# B&R Automation Studio project CleanChemi_SiteManagementSystem
Automation Studio 4.12.7.113 SP; technology packages: mapp 5.24.3, mappView 5.24.4

## Configuration 1584

### Task classes (Cpu.sw)
```
Cyclic#1 (cycle 50000 us, tolerance 50000 us):
  ModMaster <- modbusTCP.ModMaster.prg
  Main <- Main.prg
  ModbusDriv <- (binary)
Cyclic#2 (cycle 100000 us, tolerance 100000 us):
  Vis <- Vis.prg
Cyclic#4:
  Services <- Services.prg
DataObjects: Acp10sys
Binaries: FWRules, TCData, mvLoader, udbdef, TCLang, acp10cfg, arnc0cfg, Acp10map, iomap, arconfig, asfw, ashwac, sysconf, User, Role, ashwd, TC
Libraries: AsOpcUas, AsOpcUac, runtime, NcGlobal, standard, MbusTCP, IDEC_Real, astime, AsIecCon, AsTCP, AsBrStr, AsARCfg, sys_lib, ArTextSys, Str2DtPvdr, powerlnk, arssl, asstring, AsBrWStr, MpCom, MpBase, HA, HA_Version, HA_IO, HA_Dir, HA_Convert, HA_Str, HA_AlarmX, HA_ItemX, HA_RAND, ArEventLog, ArProject, brsystem, FileIO, AsUSB, HA_Array, HA_SysErr, MpAlarmX, IDEC_Strng, MpUserX, AsHttp, AsICMP, AsHost
```

### Hardware
```
X20CP1584 : X20CP1584 v1.10.0.0
  Connector IF1:
    ActivateIna = 0
  Connector IF2:
    ActivateDevice = 1
    Mode = Manual
    InternetAddress = 172.16.1.63
    SubnetMask = 255.255.255.0
    InaPort = 11160
    ActivateSnmp = 2
    ActivateModbus = 1
    NumSlaves = -1
    NumAllBlocks = -1
    MemSizeIn = -1
    MemSizeOut = -1
    SlaveDiagnostics = 1
  ConfigurationID = RemoteVis_CleanChemistry_Config1
  VolatileGlobalPvSize = 6553500
  SystemTick = 10000
  TaskClassIdleTime = 10000
  Cyclic1Duration = 50000
  Cyclic1Tolerance = 50000
  Cyclic2Duration = 100000
  Cyclic2Tolerance = 100000
  FileDevice1
  FileDeviceName1 = USER_DEVICE
  FileDevicePath1 = F:\
  FileDevice2
  FileDeviceName2 = USER_DEVICE_SIM
  FileDevicePath2 = ..\..\..\..\USER_DEVICE\
  EthernetDefaultGateway = 172.16.1.62
  ActivateDns = 1
  DnsServer1 = 8.8.8.8
  FtpUser1
  FtpUsername1 = brcpu
  FtpUserPassword1 = 20s6X0g3G25vRkBYChW+IYrxlgFH8I/njpAQzwadF+E=  // brcpu
  FtpUserSalt1 = aGb711uD
  FTPAccessRight1 = 0
  FTPdevice1 = ALL
  ActivateOpcUa = 1
  OpcUaInformationModels_PV_Version = 1
```

### Config_2.mpalarmxhistory - X20CP1584/mappServices/Config_2.mpalarmxhistory
```
Element gAlarmXHistory (Type=mpalarmxhistory)
  mapp.AlarmX.History:
    Export:
      FileNamePattern = AlarmHistory/Alarms_%Y_%m_%d_%H_%M_%S.csv
    Memory:
      MemorySize = 5
      BufferSize = 1
      MemoryType = 3
```

### Config_3.mpuserx - X20CP1584/mappServices/Config_3.mpuserx
```
Element UserMgmtX (Type=mpuserx)
  UserMgmtSystem:
    UserMgmtSystemType = 1
  ServerSettings:
    Server:
      AdditionalUserData:
        [0] = mail
        [1] = telephoneNumber
```

## Configuration 3100

CPU 5APC3100.KBU3-000, AutomationRuntime Q4.93, Build 4.1.2, Safety 0.0, Vc 

### Task classes (Cpu.sw)
```
Cyclic#1 (cycle 2000 us, tolerance 0 us):
  Master_LR <- modbusTCP.Master_LR.prg
  ModbusDriv <- (binary)
Cyclic#2 (cycle 10000 us, tolerance 10000 us):
  Vis <- Vis.prg
Cyclic#3 (cycle 100000 us, tolerance 100000 us):
  Services <- Services.prg
DataObjects: Acp10sys
Binaries: FWRules, TCData, mvLoader, udbdef, TCLang, arcoal, arflatprv, arsvcreg, iomap, arconfig, asfw, ashwac, sysconf, User, Role, ashwd, TC, Config_1, Config, Config_2, Config_3, acp10cfg, arnc0cfg, Acp10map
Libraries: AsOpcUas, AsOpcUac, runtime, NcGlobal, standard, MbusTCP, IDEC_Real, astime, AsIecCon, AsTCP, AsBrStr, AsARCfg, sys_lib, ArTextSys, Str2DtPvdr, asstring, AsBrWStr, MpCom, MpBase, HA, HA_Version, HA_IO, HA_Dir, HA_Convert, HA_AlarmX, HA_ItemX, HA_RAND, ArEventLog, ArProject, brsystem, FileIO, AsUSB, HA_Array, HA_SysErr, IDEC_Strng, MpUserX, AsHttp, AsICMP, AsHost, HA_JSON, HA_Str, ArUser, API_Login, AsIODiag, MpAlarmX, arssl, arcert, ashw, dataobj, aseth, powerlnk
```

### Hardware
```
5APC3100_KBU3_000 : 5APC3100.KBU3-000 v2.3.1.0
  Connector IF3:
    AssignedOperatingSystem = ARemb
    ActivateDevice = 1
    Mode = Manual
    InternetAddress = 172.16.1.63
    SubnetMask = 255.255.255.0
    InaPort = 11160
    ActivateSnmp = 2
    ActivateModbus = 1
    NumSlaves = -1
    NumAllBlocks = -1
    MemSizeIn = -1
    MemSizeOut = -1
  Connector IF4:
    AssignedOperatingSystem = GPOS
  Connector IF9:
    OperatingSystem = ARemb
    ActivateDevice = 1
  Connector IF5:
    AssignedOperatingSystem = GPOS
  Connector IF6:
    AssignedOperatingSystem = GPOS
  Connector IF7:
    AssignedOperatingSystem = GPOS
  Connector IF8:
    AssignedOperatingSystem = ARemb
  ConfigurationID = RemoteVis_CleanChemistry_Config1
  Simulation = 1
  VolatileGlobalPvSize = 65535000
  Connections = 10
  SystemTick = 2000
  IdleTaskClass = 3
  TaskClassIdleTime = 10000
  Cyclic1Duration = 2000
  Cyclic1Tolerance = 0
  Cyclic2Duration = 10000
  Cyclic2Tolerance = 10000
  Cyclic3Duration = 100000
  Cyclic3Tolerance = 100000
  FileDevice1
  FileDeviceName1 = USER_DEVICE
  FileDevicePath1 = F:\
  FileDevice2
  FileDeviceName2 = USER_DEVICE_SIM
  FileDevicePath2 = ..\..\..\..\USER_DEVICE\
  TimeZone = 35
  ActivateDaylightSavingTime = 1
  ActivateSntpServer = 1
  ActivateSntp = 1
  SntpcServAddr1 = time.windows.com
  EthernetDefaultGateway = 172.16.1.62
  ActivateDns = 1
  DnsServer1 = 8.8.8.8
  FtpUser1
  FtpUsername1 = brcpu
  FtpUserPassword1 = 20s6X0g3G25vRkBYChW+IYrxlgFH8I/njpAQzwadF+E=  // brcpu
  FtpUserSalt1 = aGb711uD
  FTPAccessRight1 = 0
  FTPdevice1 = ALL
  ActivateOpcUa = 1
  OpcUaLimitsMaxBrowseContinuationPoints = 10
  OpcUa_SamplingTimer1_Interval = 1000
  OpcUaInformationModels_PV_Version = 1
  ActivateHypervisor = 1
  ARembDramSizeInMb = 3072
```

### Config.mprecipexml - 5APC3100_KBU3_000/mappServices/Config.mprecipexml
```
Element gRecipeXml_Rem (Type=mprecipexml)
  mapp.Recipe.Xml:
    AutoSave = Time
      Interval = 600
      StartImmediately = FALSE
  Alarms = MpAlarmX
Element gRecipeXml_Par (Type=mprecipexml)
  Alarms = MpAlarmX
```

### Config_1.mpalarmxcore - 5APC3100_KBU3_000/mappServices/Config_1.mpalarmxcore
```
Element gAlarmXCore_HR_0 (Type=mpalarmxcore)
  mapp.AlarmX.Core:
    BySeverity:
      [0]:
        Severity = 0..100
        [0] = Reaction
          Name = SeverityAnyAlarm
      [1]:
        Severity = 0
        [0] = Reaction
          Name = Severity0
      [2]:
        Severity = 1
        [0] = Reaction
          Name = Severity1
      [3]:
        Severity = 2
        [0] = Reaction
          Name = Severity2
      [4]:
        Severity = 3
        [0] = Reaction
          Name = Severity3
      [5]:
        Severity = 4
        [0] = Reaction
          Name = Severity4
      [6]:
        Severity = 5
        [0] = Reaction
          Name = Severity5
  mapp.AlarmX.Core.Configuration:
    [0]:
      Name = RemMemLost
      Message = {$IAT/Alarm.RemMemLost}
      Code = 1
      Behavior:
        Recording:
          UnacknowledgedToAcknowledged = FALSE
    [1]:
      Name = FileLoadFailed
      Message = {$IAT/Alarm.FileLoadFailed}
      Code = 1001
      Behavior:
        Recording:
          UnacknowledgedToAcknowledged = FALSE
    [2]:
      Name = FileLoadSuccess
      Message = {$IAT/Alarm.FileLoadSuccess}
      Code = 1002
      Behavior:
        Recording:
          UnacknowledgedToAcknowledged = FALSE
    [3]:
      Name = RecipeGeneralError
      Message = {$IAT/Alarm.RecipeGeneralError}
      Code = 1003
      Behavior:
        Recording:
          UnacknowledgedToAcknowledged = FALSE
    [4]:
      Name = Severity2
      Message = {$IAT/Alarm.Severity2}
      Severity = 2
    [5]:
      Name = Severity3
      Message = {$IAT/Alarm.Severity3}
      Severity = 3
    [6]:
      Name = Severity4
      Message = {$IAT/Alarm.Severity4}
      Severity = 4
    [7]:
      Name = Severity5
      Message = {$IAT/Alarm.Severity5}
      Severity = 5
    [8]:
      Name = Severity1
      Message = {$IAT/Alarm.Severity1}
Element gAlarmXCore_LR_25 (Type=mpalarmxcore)
  mapp.AlarmX.Core:
    BySeverity:
      [0]:
        Severity = 0..100
        [0] = Reaction
          Name = SeverityAnyAlarm
      [1]:
        Severity = 0
        [0] = Reaction
          Name = Severity0
      [2]:
        Severity = 1
        [0] = Reaction
          Name = Severity1
      [3]:
        Severity = 2
        [0] = Reaction
          Name = Severity2
      [4]:
        Severity = 3
        [0] = Reaction
          Name = Severity3
      [5]:
        Severity = 4
        [0] = Reaction
          Name = Severity4
      [6]:
        Severity = 5
        [0] = Reaction
          Name = Severity5
  mapp.AlarmX.Core.Configuration:
    [0]:
      Name = RemMemLost
      Message = {$IAT/Alarm.RemMemLost}
      Code = 1
      Behavior:
        Recording:
          UnacknowledgedToAcknowledged = FALSE
    [1]:
      Name = FileLoadFailed
      Message = {$IAT/Alarm.FileLoadFailed}
      Code = 1001
      Behavior:
        Recording:
          UnacknowledgedToAcknowledged = FALSE
    [2]:
      Name = FileLoadSuccess
      Message = {$IAT/Alarm.FileLoadSuccess}
      Code = 1002
      Behavior:
        Recording:
          UnacknowledgedToAcknowledged = FALSE
    [3]:
      Name = RecipeGeneralError
      Message = {$IAT/Alarm.RecipeGeneralError}
      Code = 1003
      Behavior:
        Recording:
          UnacknowledgedToAcknowledged = FALSE
    [4]:
      Name = Severity2
      Message = {$IAT/Alarm.Severity2}
      Severity = 2
    [5]:
      Name = Severity3
      Message = {$IAT/Alarm.Severity3}
      Severity = 3
    [6]:
      Name = Severity4
      Message = {$IAT/Alarm.Severity4}
      Severity = 4
    [7]:
      Name = Severity5
      Message = {$IAT/Alarm.Severity5}
      Severity = 5
    [8]:
      Name = Severity1
      Message = {$IAT/Alarm.Severity1}
Element gAlarmXCore_LR_24 (Type=mpalarmxcore)
  mapp.AlarmX.Core:
    BySeverity:
      [0]:
        Severity = 0..100
        [0] = Reaction
          Name = SeverityAnyAlarm
      [1]:
        Severity = 0
        [0] = Reaction
          Name = Severity0
      [2]:
        Severity = 1
        [0] = Reaction
          Name = Severity1
      [3]:
        Severity = 2
        [0] = Reaction
          Name = Severity2
      [4]:
        Severity = 3
        [0] = Reaction
          Name = Severity3
      [5]:
        Severity = 4
        [0] = Reaction
          Name = Severity4
      [6]:
        Severity = 5
        [0] = Reaction
          Name = Severity5
  mapp.AlarmX.Core.Configuration:
    [0]:
      Name = RemMemLost
      Message = {$IAT/Alarm.RemMemLost}
      Code = 1
      Behavior:
        Recording:
          UnacknowledgedToAcknowledged = FALSE
    [1]:
      Name = FileLoadFailed
      Message = {$IAT/Alarm.FileLoadFailed}
      Code = 1001
      Behavior:
        Recording:
          UnacknowledgedToAcknowledged = FALSE
    [2]:
      Name = FileLoadSuccess
      Message = {$IAT/Alarm.FileLoadSuccess}
      Code = 1002
      Behavior:
        Recording:
          UnacknowledgedToAcknowledged = FALSE
    [3]:
      Name = RecipeGeneralError
      Message = {$IAT/Alarm.RecipeGeneralError}
      Code = 1003
      Behavior:
        Recording:
          UnacknowledgedToAcknowledged = FALSE
    [4]:
      Name = Severity2
      Message = {$IAT/Alarm.Severity2}
      Severity = 2
    [5]:
      Name = Severity3
      Message = {$IAT/Alarm.Severity3}
      Severity = 3
    [6]:
      Name = Severity4
      Message = {$IAT/Alarm.Severity4}
      Severity = 4
    [7]:
      Name = Severity5
      Message = {$IAT/Alarm.Severity5}
      Severity = 5
    [8]:
      Name = Severity1
      Message = {$IAT/Alarm.Severity1}
Element gAlarmXCore_LR_23 (Type=mpalarmxcore)
  mapp.AlarmX.Core:
    BySeverity:
      [0]:
        Severity = 0..100
        [0] = Reaction
          Name = SeverityAnyAlarm
      [1]:
        Severity = 0
        [0] = Reaction
          Name = Severity0
      [2]:
        Severity = 1
        [0] = Reaction
          Name = Severity1
      [3]:
        Severity = 2
        [0] = Reaction
          Name = Severity2
      [4]:
        Severity = 3
        [0] = Reaction
          Name = Severity3
      [5]:
        Severity = 4
        [0] = Reaction
          Name = Severity4
      [6]:
        Severity = 5
        [0] = Reaction
          Name = Severity5
  mapp.AlarmX.Core.Configuration:
    [0]:
      Name = RemMemLost
      Message = {$IAT/Alarm.RemMemLost}
      Code = 1
      Behavior:
        Recording:
          UnacknowledgedToAcknowledged = FALSE
    [1]:
      Name = FileLoadFailed
      Message = {$IAT/Alarm.FileLoadFailed}
      Code = 1001
      Behavior:
        Recording:
          UnacknowledgedToAcknowledged = FALSE
    [2]:
      Name = FileLoadSuccess
      Message = {$IAT/Alarm.FileLoadSuccess}
      Code = 1002
      Behavior:
        Recording:
          UnacknowledgedToAcknowledged = FALSE
    [3]:
      Name = RecipeGeneralError
      Message = {$IAT/Alarm.RecipeGeneralError}
      Code = 1003
      Behavior:
        Recording:
          UnacknowledgedToAcknowledged = FALSE
    [4]:
      Name = Severity2
      Message = {$IAT/Alarm.Severity2}
      Severity = 2
    [5]:
      Name = Severity3
      Message = {$IAT/Alarm.Severity3}
      Severity = 3
    [6]:
      Name = Severity4
      Message = {$IAT/Alarm.Severity4}
      Severity = 4
    [7]:
      Name = Severity5
      Message = {$IAT/Alarm.Severity5}
      Severity = 5
    [8]:
      Name = Severity1
      Message = {$IAT/Alarm.Severity1}
Element gAlarmXCore_LR_22 (Type=mpalarmxcore)
  mapp.AlarmX.Core:
    BySeverity:
      [0]:
        Severity = 0..100
        [0] = Reaction
          Name = SeverityAnyAlarm
      [1]:
        Severity = 0
        [0] = Reaction
          Name = Severity0
      [2]:
        Severity = 1
        [0] = Reaction
          Name = Severity1
      [3]:
        Severity = 2
        [0] = Reaction
          Name = Severity2
      [4]:
        Severity = 3
        [0] = Reaction
          Name = Severity3
      [5]:
        Severity = 4
        [0] = Reaction
          Name = Severity4
      [6]:
        Severity = 5
        [0] = Reaction
          Name = Severity5
  mapp.AlarmX.Core.Configuration:
    [0]:
      Name = RemMemLost
      Message = {$IAT/Alarm.RemMemLost}
      Code = 1
      Behavior:
        Recording:
          UnacknowledgedToAcknowledged = FALSE
    [1]:
      Name = FileLoadFailed
      Message = {$IAT/Alarm.FileLoadFailed}
      Code = 1001
      Behavior:
        Recording:
          UnacknowledgedToAcknowledged = FALSE
    [2]:
      Name = FileLoadSuccess
      Message = {$IAT/Alarm.FileLoadSuccess}
      Code = 1002
      Behavior:
        Recording:
          UnacknowledgedToAcknowledged = FALSE
    [3]:
      Name = RecipeGeneralError
      Message = {$IAT/Alarm.RecipeGeneralError}
      Code = 1003
      Behavior:
        Recording:
          UnacknowledgedToAcknowledged = FALSE
    [4]:
      Name = Severity2
      Message = {$IAT/Alarm.Severity2}
      Severity = 2
    [5]:
      Name = Severity3
      Message = {$IAT/Alarm.Severity3}
      Severity = 3
    [6]:
      Name = Severity4
      Message = {$IAT/Alarm.Severity4}
      Severity = 4
    [7]:
      Name = Severity5
      Message = {$IAT/Alarm.Severity5}
      Severity = 5
    [8]:
      Name = Severity1
      Message = {$IAT/Alarm.Severity1}
Element gAlarmXCore_LR_21 (Type=mpalarmxcore)
  mapp.AlarmX.Core:
    BySeverity:
      [0]:
        Severity = 0..100
        [0] = Reaction
          Name = SeverityAnyAlarm
      [1]:
        Severity = 0
        [0] = Reaction
          Name = Severity0
      [2]:
        Severity = 1
        [0] = Reaction
          Name = Severity1
      [3]:
        Severity = 2
        [0] = Reaction
          Name = Severity2
      [4]:
        Severity = 3
        [0] = Reaction
          Name = Severity3
      [5]:
        Severity = 4
        [0] = Reaction
          Name = Severity4
      [6]:
        Severity = 5
        [0] = Reaction
          Name = Severity5
  mapp.AlarmX.Core.Configuration:
    [0]:
      Name = RemMemLost
      Message = {$IAT/Alarm.RemMemLost}
      Code = 1
      Behavior:
        Recording:
          UnacknowledgedToAcknowledged = FALSE
    [1]:
      Name = FileLoadFailed
      Message = {$IAT/Alarm.FileLoadFailed}
      Code = 1001
      Behavior:
        Recording:
          UnacknowledgedToAcknowledged = FALSE
    [2]:
      Name = FileLoadSuccess
      Message = {$IAT/Alarm.FileLoadSuccess}
      Code = 1002
      Behavior:
        Recording:
          UnacknowledgedToAcknowledged = FALSE
    [3]:
      Name = RecipeGeneralError
      Message = {$IAT/Alarm.RecipeGeneralError}
      Code = 1003
      Behavior:
        Recording:
          UnacknowledgedToAcknowledged = FALSE
    [4]:
      Name = Severity2
      Message = {$IAT/Alarm.Severity2}
      Severity = 2
    [5]:
      Name = Severity3
      Message = {$IAT/Alarm.Severity3}
      Severity = 3
    [6]:
      Name = Severity4
      Message = {$IAT/Alarm.Severity4}
      Severity = 4
    [7]:
      Name = Severity5
      Message = {$IAT/Alarm.Severity5}
      Severity = 5
    [8]:
      Name = Severity1
      Message = {$IAT/Alarm.Severity1}
Element gAlarmXCore_LR_20 (Type=mpalarmxcore)
  mapp.AlarmX.Core:
    BySeverity:
      [0]:
        Severity = 0..100
        [0] = Reaction
          Name = SeverityAnyAlarm
      [1]:
        Severity = 0
        [0] = Reaction
          Name = Severity0
      [2]:
        Severity = 1
        [0] = Reaction
          Name = Severity1
      [3]:
        Severity = 2
        [0] = Reaction
          Name = Severity2
      [4]:
        Severity = 3
        [0] = Reaction
          Name = Severity3
      [5]:
        Severity = 4
        [0] = Reaction
          Name = Severity4
      [6]:
        Severity = 5
        [0] = Reaction
          Name = Severity5
  mapp.AlarmX.Core.Configuration:
    [0]:
      Name = RemMemLost
      Message = {$IAT/Alarm.RemMemLost}
      Code = 1
      Behavior:
        Recording:
          UnacknowledgedToAcknowledged = FALSE
    [1]:
      Name = FileLoadFailed
      Message = {$IAT/Alarm.FileLoadFailed}
      Code = 1001
      Behavior:
        Recording:
          UnacknowledgedToAcknowledged = FALSE
    [2]:
      Name = FileLoadSuccess
      Message = {$IAT/Alarm.FileLoadSuccess}
      Code = 1002
      Behavior:
        Recording:
          UnacknowledgedToAcknowledged = FALSE
    [3]:
      Name = RecipeGeneralError
      Message = {$IAT/Alarm.RecipeGeneralError}
      Code = 1003
      Behavior:
        Recording:
          UnacknowledgedToAcknowledged = FALSE
    [4]:
      Name = Severity2
      Message = {$IAT/Alarm.Severity2}
      Severity = 2
    [5]:
      Name = Severity3
      Message = {$IAT/Alarm.Severity3}
      Severity = 3
    [6]:
      Name = Severity4
      Message = {$IAT/Alarm.Severity4}
      Severity = 4
    [7]:
      Name = Severity5
      Message = {$IAT/Alarm.Severity5}
      Severity = 5
    [8]:
      Name = Severity1
      Message = {$IAT/Alarm.Severity1}
Element gAlarmXCore_LR_19 (Type=mpalarmxcore)
  mapp.AlarmX.Core:
    BySeverity:
      [0]:
        Severity = 0..100
        [0] = Reaction
          Name = SeverityAnyAlarm
      [1]:
        Severity = 0
        [0] = Reaction
          Name = Severity0
      [2]:
        Severity = 1
        [0] = Reaction
          Name = Severity1
      [3]:
        Severity = 2
        [0] = Reaction
          Name = Severity2
      [4]:
        Severity = 3
        [0] = Reaction
          Name = Severity3
      [5]:
        Severity = 4
        [0] = Reaction
          Name = Severity4
      [6]:
        Severity = 5
        [0] = Reaction
          Name = Severity5
  mapp.AlarmX.Core.Configuration:
    [0]:
      Name = RemMemLost
      Message = {$IAT/Alarm.RemMemLost}
      Code = 1
      Behavior:
        Recording:
          UnacknowledgedToAcknowledged = FALSE
    [1]:
      Name = FileLoadFailed
      Message = {$IAT/Alarm.FileLoadFailed}
      Code = 1001
      Behavior:
        Recording:
          UnacknowledgedToAcknowledged = FALSE
    [2]:
      Name = FileLoadSuccess
      Message = {$IAT/Alarm.FileLoadSuccess}
      Code = 1002
      Behavior:
        Recording:
          UnacknowledgedToAcknowledged = FALSE
    [3]:
      Name = RecipeGeneralError
      Message = {$IAT/Alarm.RecipeGeneralError}
      Code = 1003
      Behavior:
        Recording:
          UnacknowledgedToAcknowledged = FALSE
    [4]:
      Name = Severity2
      Message = {$IAT/Alarm.Severity2}
      Severity = 2
    [5]:
      Name = Severity3
      Message = {$IAT/Alarm.Severity3}
      Severity = 3
    [6]:
      Name = Severity4
      Message = {$IAT/Alarm.Severity4}
      Severity = 4
    [7]:
      Name = Severity5
      Message = {$IAT/Alarm.Severity5}
      Severity = 5
    [8]:
      Name = Severity1
      Message = {$IAT/Alarm.Severity1}
Element gAlarmXCore_LR_18 (Type=mpalarmxcore)
  mapp.AlarmX.Core:
    BySeverity:
      [0]:
        Severity = 0..100
        [0] = Reaction
          Name = SeverityAnyAlarm
      [1]:
        Severity = 0
        [0] = Reaction
          Name = Severity0
      [2]:
        Severity = 1
        [0] = Reaction
          Name = Severity1
      [3]:
        Severity = 2
        [0] = Reaction
          Name = Severity2
      [4]:
        Severity = 3
        [0] = Reaction
          Name = Severity3
      [5]:
        Severity = 4
        [0] = Reaction
          Name = Severity4
      [6]:
        Severity = 5
        [0] = Reaction
          Name = Severity5
  mapp.AlarmX.Core.Configuration:
    [0]:
      Name = RemMemLost
      Message = {$IAT/Alarm.RemMemLost}
      Code = 1
      Behavior:
        Recording:
          UnacknowledgedToAcknowledged = FALSE
    [1]:
      Name = FileLoadFailed
      Message = {$IAT/Alarm.FileLoadFailed}
      Code = 1001
      Behavior:
        Recording:
          UnacknowledgedToAcknowledged = FALSE
    [2]:
      Name = FileLoadSuccess
      Message = {$IAT/Alarm.FileLoadSuccess}
      Code = 1002
      Behavior:
        Recording:
          UnacknowledgedToAcknowledged = FALSE
    [3]:
      Name = RecipeGeneralError
      Message = {$IAT/Alarm.RecipeGeneralError}
      Code = 1003
      Behavior:
        Recording:
          UnacknowledgedToAcknowledged = FALSE
    [4]:
      Name = Severity2
      Message = {$IAT/Alarm.Severity2}
      Severity = 2
    [5]:
      Name = Severity3
      Message = {$IAT/Alarm.Severity3}
      Severity = 3
    [6]:
      Name = Severity4
      Message = {$IAT/Alarm.Severity4}
      Severity = 4
    [7]:
      Name = Severity5
      Message = {$IAT/Alarm.Severity5}
      Severity = 5
    [8]:
      Name = Severity1
      Message = {$IAT/Alarm.Severity1}
Element gAlarmXCore_LR_17 (Type=mpalarmxcore)
  mapp.AlarmX.Core:
    BySeverity:
      [0]:
        Severity = 0..100
        [0] = Reaction
          Name = SeverityAnyAlarm
      [1]:
        Severity = 0
        [0] = Reaction
          Name = Severity0
      [2]:
        Severity = 1
        [0] = Reaction
          Name = Severity1
      [3]:
        Severity = 2
        [0] = Reaction
          Name = Severity2
      [4]:
        Severity = 3
        [0] = Reaction
          Name = Severity3
      [5]:
        Severity = 4
        [0] = Reaction
          Name = Severity4
      [6]:
        Severity = 5
        [0] = Reaction
          Name = Severity5
  mapp.AlarmX.Core.Configuration:
    [0]:
      Name = RemMemLost
      Message = {$IAT/Alarm.RemMemLost}
      Code = 1
      Behavior:
        Recording:
          UnacknowledgedToAcknowledged = FALSE
    [1]:
      Name = FileLoadFailed
      Message = {$IAT/Alarm.FileLoadFailed}
      Code = 1001
      Behavior:
        Recording:
          UnacknowledgedToAcknowledged = FALSE
    [2]:
      Name = FileLoadSuccess
      Message = {$IAT/Alarm.FileLoadSuccess}
      Code = 1002
      Behavior:
        Recording:
          UnacknowledgedToAcknowledged = FALSE
    [3]:
      Name = RecipeGeneralError
      Message = {$IAT/Alarm.RecipeGeneralError}
      Code = 1003
      Behavior:
        Recording:
          UnacknowledgedToAcknowledged = FALSE
    [4]:
      Name = Severity2
      Message = {$IAT/Alarm.Severity2}
      Severity = 2
    [5]:
      Name = Severity3
      Message = {$IAT/Alarm.Severity3}
      Severity = 3
    [6]:
      Name = Severity4
      Message = {$IAT/Alarm.Severity4}
      Severity = 4
    [7]:
      Name = Severity5
      Message = {$IAT/Alarm.Severity5}
      Severity = 5
    [8]:
      Name = Severity1
      Message = {$IAT/Alarm.Severity1}
Element gAlarmXCore_LR_16 (Type=mpalarmxcore)
  mapp.AlarmX.Core:
    BySeverity:
      [0]:
        Severity = 0..100
        [0] = Reaction
          Name = SeverityAnyAlarm
      [1]:
        Severity = 0
        [0] = Reaction
          Name = Severity0
      [2]:
        Severity = 1
        [0] = Reaction
          Name = Severity1
      [3]:
        Severity = 2
        [0] = Reaction
          Name = Severity2
      [4]:
        Severity = 3
        [0] = Reaction
          Name = Severity3
      [5]:
        Severity = 4
        [0] = Reaction
          Name = Severity4
      [6]:
        Severity = 5
        [0] = Reaction
          Name = Severity5
  mapp.AlarmX.Core.Configuration:
    [0]:
      Name = RemMemLost
      Message = {$IAT/Alarm.RemMemLost}
      Code = 1
      Behavior:
        Recording:
          UnacknowledgedToAcknowledged = FALSE
    [1]:
      Name = FileLoadFailed
      Message = {$IAT/Alarm.FileLoadFailed}
      Code = 1001
      Behavior:
        Recording:
          UnacknowledgedToAcknowledged = FALSE
    [2]:
      Name = FileLoadSuccess
      Message = {$IAT/Alarm.FileLoadSuccess}
      Code = 1002
      Behavior:
        Recording:
          UnacknowledgedToAcknowledged = FALSE
    [3]:
      Name = RecipeGeneralError
      Message = {$IAT/Alarm.RecipeGeneralError}
      Code = 1003
      Behavior:
        Recording:
          UnacknowledgedToAcknowledged = FALSE
    [4]:
      Name = Severity2
      Message = {$IAT/Alarm.Severity2}
      Severity = 2
    [5]:
      Name = Severity3
      Message = {$IAT/Alarm.Severity3}
      Severity = 3
    [6]:
      Name = Severity4
      Message = {$IAT/Alarm.Severity4}
      Severity = 4
    [7]:
      Name = Severity5
      Message = {$IAT/Alarm.Severity5}
      Severity = 5
    [8]:
      Name = Severity1
      Message = {$IAT/Alarm.Severity1}
Element gAlarmXCore_LR_15 (Type=mpalarmxcore)
  mapp.AlarmX.Core:
    BySeverity:
      [0]:
        Severity = 0..100
        [0] = Reaction
          Name = SeverityAnyAlarm
      [1]:
        Severity = 0
        [0] = Reaction
          Name = Severity0
      [2]:
        Severity = 1
        [0] = Reaction
          Name = Severity1
      [3]:
        Severity = 2
        [0] = Reaction
          Name = Severity2
      [4]:
        Severity = 3
        [0] = Reaction
          Name = Severity3
      [5]:
        Severity = 4
        [0] = Reaction
          Name = Severity4
      [6]:
        Severity = 5
        [0] = Reaction
          Name = Severity5
  mapp.AlarmX.Core.Configuration:
    [0]:
      Name = RemMemLost
      Message = {$IAT/Alarm.RemMemLost}
      Code = 1
      Behavior:
        Recording:
          UnacknowledgedToAcknowledged = FALSE
    [1]:
      Name = FileLoadFailed
      Message = {$IAT/Alarm.FileLoadFailed}
      Code = 1001
      Behavior:
        Recording:
          UnacknowledgedToAcknowledged = FALSE
    [2]:
      Name = FileLoadSuccess
      Message = {$IAT/Alarm.FileLoadSuccess}
      Code = 1002
      Behavior:
        Recording:
          UnacknowledgedToAcknowledged = FALSE
    [3]:
      Name = RecipeGeneralError
      Message = {$IAT/Alarm.RecipeGeneralError}
      Code = 1003
      Behavior:
        Recording:
          UnacknowledgedToAcknowledged = FALSE
    [4]:
      Name = Severity2
      Message = {$IAT/Alarm.Severity2}
      Severity = 2
    [5]:
      Name = Severity3
      Message = {$IAT/Alarm.Severity3}
      Severity = 3
    [6]:
      Name = Severity4
      Message = {$IAT/Alarm.Severity4}
      Severity = 4
    [7]:
      Name = Severity5
      Message = {$IAT/Alarm.Severity5}
      Severity = 5
    [8]:
      Name = Severity1
      Message = {$IAT/Alarm.Severity1}
Element gAlarmXCore_LR_14 (Type=mpalarmxcore)
  mapp.AlarmX.Core:
    BySeverity:
      [0]:
        Severity = 0..100
        [0] = Reaction
          Name = SeverityAnyAlarm
      [1]:
        Severity = 0
        [0] = Reaction
          Name = Severity0
      [2]:
        Severity = 1
        [0] = Reaction
          Name = Severity1
      [3]:
        Severity = 2
        [0] = Reaction
          Name = Severity2
      [4]:
        Severity = 3
        [0] = Reaction
          Name = Severity3
      [5]:
        Severity = 4
        [0] = Reaction
          Name = Severity4
      [6]:
        Severity = 5
        [0] = Reaction
          Name = Severity5
  mapp.AlarmX.Core.Configuration:
    [0]:
      Name = RemMemLost
      Message = {$IAT/Alarm.RemMemLost}
      Code = 1
      Behavior:
        Recording:
          UnacknowledgedToAcknowledged = FALSE
    [1]:
      Name = FileLoadFailed
      Message = {$IAT/Alarm.FileLoadFailed}
      Code = 1001
      Behavior:
        Recording:
          UnacknowledgedToAcknowledged = FALSE
    [2]:
      Name = FileLoadSuccess
      Message = {$IAT/Alarm.FileLoadSuccess}
      Code = 1002
      Behavior:
        Recording:
          UnacknowledgedToAcknowledged = FALSE
    [3]:
      Name = RecipeGeneralError
      Message = {$IAT/Alarm.RecipeGeneralError}
      Code = 1003
      Behavior:
        Recording:
          UnacknowledgedToAcknowledged = FALSE
    [4]:
      Name = Severity2
      Message = {$IAT/Alarm.Severity2}
      Severity = 2
    [5]:
      Name = Severity3
      Message = {$IAT/Alarm.Severity3}
      Severity = 3
    [6]:
      Name = Severity4
      Message = {$IAT/Alarm.Severity4}
      Severity = 4
    [7]:
      Name = Severity5
      Message = {$IAT/Alarm.Severity5}
      Severity = 5
    [8]:
      Name = Severity1
      Message = {$IAT/Alarm.Severity1}
Element gAlarmXCore_LR_13 (Type=mpalarmxcore)
  mapp.AlarmX.Core:
    BySeverity:
      [0]:
        Severity = 0..100
        [0] = Reaction
          Name = SeverityAnyAlarm
      [1]:
        Severity = 0
        [0] = Reaction
          Name = Severity0
      [2]:
        Severity = 1
        [0] = Reaction
          Name = Severity1
      [3]:
        Severity = 2
        [0] = Reaction
          Name = Severity2
      [4]:
        Severity = 3
        [0] = Reaction
          Name = Severity3
      [5]:
        Severity = 4
        [0] = Reaction
          Name = Severity4
      [6]:
        Severity = 5
        [0] = Reaction
          Name = Severity5
  mapp.AlarmX.Core.Configuration:
    [0]:
      Name = RemMemLost
      Message = {$IAT/Alarm.RemMemLost}
      Code = 1
      Behavior:
        Recording:
          UnacknowledgedToAcknowledged = FALSE
    [1]:
      Name = FileLoadFailed
      Message = {$IAT/Alarm.FileLoadFailed}
      Code = 1001
      Behavior:
        Recording:
          UnacknowledgedToAcknowledged = FALSE
    [2]:
      Name = FileLoadSuccess
      Message = {$IAT/Alarm.FileLoadSuccess}
      Code = 1002
      Behavior:
        Recording:
          UnacknowledgedToAcknowledged = FALSE
    [3]:
      Name = RecipeGeneralError
      Message = {$IAT/Alarm.RecipeGeneralError}
      Code = 1003
      Behavior:
        Recording:
          UnacknowledgedToAcknowledged = FALSE
    [4]:
      Name = Severity2
      Message = {$IAT/Alarm.Severity2}
      Severity = 2
    [5]:
      Name = Severity3
      Message = {$IAT/Alarm.Severity3}
      Severity = 3
    [6]:
      Name = Severity4
      Message = {$IAT/Alarm.Severity4}
      Severity = 4
    [7]:
      Name = Severity5
      Message = {$IAT/Alarm.Severity5}
      Severity = 5
    [8]:
      Name = Severity1
      Message = {$IAT/Alarm.Severity1}
Element gAlarmXCore_LR_12 (Type=mpalarmxcore)
  mapp.AlarmX.Core:
    BySeverity:
      [0]:
        Severity = 0..100
        [0] = Reaction
          Name = SeverityAnyAlarm
      [1]:
        Severity = 0
        [0] = Reaction
          Name = Severity0
      [2]:
        Severity = 1
        [0] = Reaction
          Name = Severity1
      [3]:
        Severity = 2
        [0] = Reaction
          Name = Severity2
      [4]:
        Severity = 3
        [0] = Reaction
          Name = Severity3
      [5]:
        Severity = 4
        [0] = Reaction
          Name = Severity4
      [6]:
        Severity = 5
        [0] = Reaction
          Name = Severity5
  mapp.AlarmX.Core.Configuration:
    [0]:
      Name = RemMemLost
      Message = {$IAT/Alarm.RemMemLost}
      Code = 1
      Behavior:
        Recording:
          UnacknowledgedToAcknowledged = FALSE
    [1]:
      Name = FileLoadFailed
      Message = {$IAT/Alarm.FileLoadFailed}
      Code = 1001
      Behavior:
        Recording:
          UnacknowledgedToAcknowledged = FALSE
    [2]:
      Name = FileLoadSuccess
      Message = {$IAT/Alarm.FileLoadSuccess}
      Code = 1002
      Behavior:
        Recording:
          UnacknowledgedToAcknowledged = FALSE
    [3]:
      Name = RecipeGeneralError
      Message = {$IAT/Alarm.RecipeGeneralError}
      Code = 1003
      Behavior:
        Recording:
          UnacknowledgedToAcknowledged = FALSE
    [4]:
      Name = Severity2
      Message = {$IAT/Alarm.Severity2}
      Severity = 2
    [5]:
      Name = Severity3
      Message = {$IAT/Alarm.Severity3}
      Severity = 3
    [6]:
      Name = Severity4
      Message = {$IAT/Alarm.Severity4}
      Severity = 4
    [7]:
      Name = Severity5
      Message = {$IAT/Alarm.Severity5}
      Severity = 5
    [8]:
      Name = Severity1
      Message = {$IAT/Alarm.Severity1}
Element gAlarmXCore_LR_11 (Type=mpalarmxcore)
  mapp.AlarmX.Core:
    BySeverity:
      [0]:
        Severity = 0..100
        [0] = Reaction
          Name = SeverityAnyAlarm
      [1]:
        Severity = 0
        [0] = Reaction
          Name = Severity0
      [2]:
        Severity = 1
        [0] = Reaction
          Name = Severity1
      [3]:
        Severity = 2
        [0] = Reaction
          Name = Severity2
      [4]:
        Severity = 3
        [0] = Reaction
          Name = Severity3
      [5]:
        Severity = 4
        [0] = Reaction
          Name = Severity4
      [6]:
        Severity = 5
        [0] = Reaction
          Name = Severity5
  mapp.AlarmX.Core.Configuration:
    [0]:
      Name = RemMemLost
      Message = {$IAT/Alarm.RemMemLost}
      Code = 1
      Behavior:
        Recording:
          UnacknowledgedToAcknowledged = FALSE
    [1]:
      Name = FileLoadFailed
      Message = {$IAT/Alarm.FileLoadFailed}
      Code = 1001
      Behavior:
        Recording:
          UnacknowledgedToAcknowledged = FALSE
    [2]:
      Name = FileLoadSuccess
      Message = {$IAT/Alarm.FileLoadSuccess}
      Code = 1002
      Behavior:
        Recording:
          UnacknowledgedToAcknowledged = FALSE
    [3]:
      Name = RecipeGeneralError
      Message = {$IAT/Alarm.RecipeGeneralError}
      Code = 1003
      Behavior:
        Recording:
          UnacknowledgedToAcknowledged = FALSE
    [4]:
      Name = Severity2
      Message = {$IAT/Alarm.Severity2}
      Severity = 2
    [5]:
      Name = Severity3
      Message = {$IAT/Alarm.Severity3}
      Severity = 3
    [6]:
      Name = Severity4
      Message = {$IAT/Alarm.Severity4}
      Severity = 4
    [7]:
      Name = Severity5
      Message = {$IAT/Alarm.Severity5}
      Severity = 5
    [8]:
      Name = Severity1
      Message = {$IAT/Alarm.Severity1}
Element gAlarmXCore_LR_10 (Type=mpalarmxcore)
  mapp.AlarmX.Core:
    BySeverity:
      [0]:
        Severity = 0..100
        [0] = Reaction
          Name = SeverityAnyAlarm
      [1]:
        Severity = 0
        [0] = Reaction
          Name = Severity0
      [2]:
        Severity = 1
        [0] = Reaction
          Name = Severity1
      [3]:
        Severity = 2
        [0] = Reaction
          Name = Severity2
      [4]:
        Severity = 3
        [0] = Reaction
          Name = Severity3
      [5]:
        Severity = 4
        [0] = Reaction
          Name = Severity4
      [6]:
        Severity = 5
        [0] = Reaction
          Name = Severity5
  mapp.AlarmX.Core.Configuration:
    [0]:
      Name = RemMemLost
      Message = {$IAT/Alarm.RemMemLost}
      Code = 1
      Behavior:
        Recording:
          UnacknowledgedToAcknowledged = FALSE
    [1]:
      Name = FileLoadFailed
      Message = {$IAT/Alarm.FileLoadFailed}
      Code = 1001
      Behavior:
        Recording:
          UnacknowledgedToAcknowledged = FALSE
    [2]:
      Name = FileLoadSuccess
      Message = {$IAT/Alarm.FileLoadSuccess}
      Code = 1002
      Behavior:
        Recording:
          UnacknowledgedToAcknowledged = FALSE
    [3]:
      Name = RecipeGeneralError
      Message = {$IAT/Alarm.RecipeGeneralError}
      Code = 1003
      Behavior:
        Recording:
          UnacknowledgedToAcknowledged = FALSE
    [4]:
      Name = Severity2
      Message = {$IAT/Alarm.Severity2}
      Severity = 2
    [5]:
      Name = Severity3
      Message = {$IAT/Alarm.Severity3}
      Severity = 3
    [6]:
      Name = Severity4
      Message = {$IAT/Alarm.Severity4}
      Severity = 4
    [7]:
      Name = Severity5
      Message = {$IAT/Alarm.Severity5}
      Severity = 5
    [8]:
      Name = Severity1
      Message = {$IAT/Alarm.Severity1}
Element gAlarmXCore_LR_9 (Type=mpalarmxcore)
  mapp.AlarmX.Core:
    BySeverity:
      [0]:
        Severity = 0..100
        [0] = Reaction
          Name = SeverityAnyAlarm
      [1]:
        Severity = 0
        [0] = Reaction
          Name = Severity0
      [2]:
        Severity = 1
        [0] = Reaction
          Name = Severity1
      [3]:
        Severity = 2
        [0] = Reaction
          Name = Severity2
      [4]:
        Severity = 3
        [0] = Reaction
          Name = Severity3
      [5]:
        Severity = 4
        [0] = Reaction
          Name = Severity4
      [6]:
        Severity = 5
        [0] = Reaction
          Name = Severity5
  mapp.AlarmX.Core.Configuration:
    [0]:
      Name = RemMemLost
      Message = {$IAT/Alarm.RemMemLost}
      Code = 1
      Behavior:
        Recording:
          UnacknowledgedToAcknowledged = FALSE
    [1]:
      Name = FileLoadFailed
      Message = {$IAT/Alarm.FileLoadFailed}
      Code = 1001
      Behavior:
        Recording:
          UnacknowledgedToAcknowledged = FALSE
    [2]:
      Name = FileLoadSuccess
      Message = {$IAT/Alarm.FileLoadSuccess}
      Code = 1002
      Behavior:
        Recording:
          UnacknowledgedToAcknowledged = FALSE
    [3]:
      Name = RecipeGeneralError
      Message = {$IAT/Alarm.RecipeGeneralError}
      Code = 1003
      Behavior:
        Recording:
          UnacknowledgedToAcknowledged = FALSE
    [4]:
      Name = Severity2
      Message = {$IAT/Alarm.Severity2}
      Severity = 2
    [5]:
      Name = Severity3
      Message = {$IAT/Alarm.Severity3}
      Severity = 3
    [6]:
      Name = Severity4
      Message = {$IAT/Alarm.Severity4}
      Severity = 4
    [7]:
      Name = Severity5
      Message = {$IAT/Alarm.Severity5}
      Severity = 5
    [8]:
      Name = Severity1
      Message = {$IAT/Alarm.Severity1}
Element gAlarmXCore_LR_8 (Type=mpalarmxcore)
  mapp.AlarmX.Core:
    BySeverity:
      [0]:
        Severity = 0..100
        [0] = Reaction
          Name = SeverityAnyAlarm
      [1]:
        Severity = 0
        [0] = Reaction
          Name = Severity0
      [2]:
        Severity = 1
        [0] = Reaction
          Name = Severity1
      [3]:
        Severity = 2
        [0] = Reaction
          Name = Severity2
      [4]:
        Severity = 3
        [0] = Reaction
          Name = Severity3
      [5]:
        Severity = 4
        [0] = Reaction
          Name = Severity4
      [6]:
        Severity = 5
        [0] = Reaction
          Name = Severity5
  mapp.AlarmX.Core.Configuration:
    [0]:
      Name = RemMemLost
      Message = {$IAT/Alarm.RemMemLost}
      Code = 1
      Behavior:
        Recording:
          UnacknowledgedToAcknowledged = FALSE
    [1]:
      Name = FileLoadFailed
      Message = {$IAT/Alarm.FileLoadFailed}
      Code = 1001
      Behavior:
        Recording:
          UnacknowledgedToAcknowledged = FALSE
    [2]:
      Name = FileLoadSuccess
      Message = {$IAT/Alarm.FileLoadSuccess}
      Code = 1002
      Behavior:
        Recording:
          UnacknowledgedToAcknowledged = FALSE
    [3]:
      Name = RecipeGeneralError
      Message = {$IAT/Alarm.RecipeGeneralError}
      Code = 1003
      Behavior:
        Recording:
          UnacknowledgedToAcknowledged = FALSE
    [4]:
      Name = Severity2
      Message = {$IAT/Alarm.Severity2}
      Severity = 2
    [5]:
      Name = Severity3
      Message = {$IAT/Alarm.Severity3}
      Severity = 3
    [6]:
      Name = Severity4
      Message = {$IAT/Alarm.Severity4}
      Severity = 4
    [7]:
      Name = Severity5
      Message = {$IAT/Alarm.Severity5}
      Severity = 5
    [8]:
      Name = Severity1
      Message = {$IAT/Alarm.Severity1}
Element gAlarmXCore_LR_7 (Type=mpalarmxcore)
  mapp.AlarmX.Core:
    BySeverity:
      [0]:
        Severity = 0..100
        [0] = Reaction
          Name = SeverityAnyAlarm
      [1]:
        Severity = 0
        [0] = Reaction
          Name = Severity0
      [2]:
        Severity = 1
        [0] = Reaction
          Name = Severity1
      [3]:
        Severity = 2
        [0] = Reaction
          Name = Severity2
      [4]:
        Severity = 3
        [0] = Reaction
          Name = Severity3
      [5]:
        Severity = 4
        [0] = Reaction
          Name = Severity4
      [6]:
        Severity = 5
        [0] = Reaction
          Name = Severity5
  mapp.AlarmX.Core.Configuration:
    [0]:
      Name = RemMemLost
      Message = {$IAT/Alarm.RemMemLost}
      Code = 1
      Behavior:
        Recording:
          UnacknowledgedToAcknowledged = FALSE
    [1]:
      Name = FileLoadFailed
      Message = {$IAT/Alarm.FileLoadFailed}
      Code = 1001
      Behavior:
        Recording:
          UnacknowledgedToAcknowledged = FALSE
    [2]:
      Name = FileLoadSuccess
      Message = {$IAT/Alarm.FileLoadSuccess}
      Code = 1002
      Behavior:
        Recording:
          UnacknowledgedToAcknowledged = FALSE
    [3]:
      Name = RecipeGeneralError
      Message = {$IAT/Alarm.RecipeGeneralError}
      Code = 1003
      Behavior:
        Recording:
          UnacknowledgedToAcknowledged = FALSE
    [4]:
      Name = Severity2
      Message = {$IAT/Alarm.Severity2}
      Severity = 2
    [5]:
      Name = Severity3
      Message = {$IAT/Alarm.Severity3}
      Severity = 3
    [6]:
      Name = Severity4
      Message = {$IAT/Alarm.Severity4}
      Severity = 4
    [7]:
      Name = Severity5
      Message = {$IAT/Alarm.Severity5}
      Severity = 5
    [8]:
      Name = Severity1
      Message = {$IAT/Alarm.Severity1}
Element gAlarmXCore_LR_5 (Type=mpalarmxcore)
  mapp.AlarmX.Core:
    BySeverity:
      [0]:
        Severity = 0..100
        [0] = Reaction
          Name = SeverityAnyAlarm
      [1]:
        Severity = 0
        [0] = Reaction
          Name = Severity0
      [2]:
        Severity = 1
        [0] = Reaction
          Name = Severity1
      [3]:
        Severity = 2
        [0] = Reaction
          Name = Severity2
      [4]:
        Severity = 3
        [0] = Reaction
          Name = Severity3
      [5]:
        Severity = 4
        [0] = Reaction
          Name = Severity4
      [6]:
        Severity = 5
        [0] = Reaction
          Name = Severity5
  mapp.AlarmX.Core.Configuration:
    [0]:
      Name = RemMemLost
      Message = {$IAT/Alarm.RemMemLost}
      Code = 1
      Behavior:
        Recording:
          UnacknowledgedToAcknowledged = FALSE
    [1]:
      Name = FileLoadFailed
      Message = {$IAT/Alarm.FileLoadFailed}
      Code = 1001
      Behavior:
        Recording:
          UnacknowledgedToAcknowledged = FALSE
    [2]:
      Name = FileLoadSuccess
      Message = {$IAT/Alarm.FileLoadSuccess}
      Code = 1002
      Behavior:
        Recording:
          UnacknowledgedToAcknowledged = FALSE
    [3]:
      Name = RecipeGeneralError
      Message = {$IAT/Alarm.RecipeGeneralError}
      Code = 1003
      Behavior:
        Recording:
          UnacknowledgedToAcknowledged = FALSE
    [4]:
      Name = Severity2
      Message = {$IAT/Alarm.Severity2}
      Severity = 2
    [5]:
      Name = Severity3
      Message = {$IAT/Alarm.Severity3}
      Severity = 3
    [6]:
      Name = Severity4
      Message = {$IAT/Alarm.Severity4}
      Severity = 4
    [7]:
      Name = Severity5
      Message = {$IAT/Alarm.Severity5}
      Severity = 5
    [8]:
      Name = Severity1
      Message = {$IAT/Alarm.Severity1}
Element gAlarmXCore_LR_6 (Type=mpalarmxcore)
  mapp.AlarmX.Core:
    BySeverity:
      [0]:
        Severity = 0..100
        [0] = Reaction
          Name = SeverityAnyAlarm
      [1]:
        Severity = 0
        [0] = Reaction
          Name = Severity0
      [2]:
        Severity = 1
        [0] = Reaction
          Name = Severity1
      [3]:
        Severity = 2
        [0] = Reaction
          Name = Severity2
      [4]:
        Severity = 3
        [0] = Reaction
          Name = Severity3
      [5]:
        Severity = 4
        [0] = Reaction
          Name = Severity4
      [6]:
        Severity = 5
        [0] = Reaction
          Name = Severity5
  mapp.AlarmX.Core.Configuration:
    [0]:
      Name = RemMemLost
      Message = {$IAT/Alarm.RemMemLost}
      Code = 1
      Behavior:
        Recording:
          UnacknowledgedToAcknowledged = FALSE
    [1]:
      Name = FileLoadFailed
      Message = {$IAT/Alarm.FileLoadFailed}
      Code = 1001
      Behavior:
        Recording:
          UnacknowledgedToAcknowledged = FALSE
    [2]:
      Name = FileLoadSuccess
      Message = {$IAT/Alarm.FileLoadSuccess}
      Code = 1002
      Behavior:
        Recording:
          UnacknowledgedToAcknowledged = FALSE
    [3]:
      Name = RecipeGeneralError
      Message = {$IAT/Alarm.RecipeGeneralError}
      Code = 1003
      Behavior:
        Recording:
          UnacknowledgedToAcknowledged = FALSE
    [4]:
      Name = Severity2
      Message = {$IAT/Alarm.Severity2}
      Severity = 2
    [5]:
      Name = Severity3
      Message = {$IAT/Alarm.Severity3}
      Severity = 3
    [6]:
      Name = Severity4
      Message = {$IAT/Alarm.Severity4}
      Severity = 4
    [7]:
      Name = Severity5
      Message = {$IAT/Alarm.Severity5}
      Severity = 5
    [8]:
      Name = Severity1
      Message = {$IAT/Alarm.Severity1}
Element gAlarmXCore_LR_4 (Type=mpalarmxcore)
  mapp.AlarmX.Core:
    BySeverity:
      [0]:
        Severity = 0..100
        [0] = Reaction
          Name = SeverityAnyAlarm
      [1]:
        Severity = 0
        [0] = Reaction
          Name = Severity0
      [2]:
        Severity = 1
        [0] = Reaction
          Name = Severity1
      [3]:
        Severity = 2
        [0] = Reaction
          Name = Severity2
      [4]:
        Severity = 3
        [0] = Reaction
          Name = Severity3
      [5]:
        Severity = 4
        [0] = Reaction
          Name = Severity4
      [6]:
        Severity = 5
        [0] = Reaction
          Name = Severity5
  mapp.AlarmX.Core.Configuration:
    [0]:
      Name = RemMemLost
      Message = {$IAT/Alarm.RemMemLost}
      Code = 1
      Behavior:
        Recording:
          UnacknowledgedToAcknowledged = FALSE
    [1]:
      Name = FileLoadFailed
      Message = {$IAT/Alarm.FileLoadFailed}
      Code = 1001
      Behavior:
        Recording:
          UnacknowledgedToAcknowledged = FALSE
    [2]:
      Name = FileLoadSuccess
      Message = {$IAT/Alarm.FileLoadSuccess}
      Code = 1002
      Behavior:
        Recording:
          UnacknowledgedToAcknowledged = FALSE
    [3]:
      Name = RecipeGeneralError
      Message = {$IAT/Alarm.RecipeGeneralError}
      Code = 1003
      Behavior:
        Recording:
          UnacknowledgedToAcknowledged = FALSE
    [4]:
      Name = Severity2
      Message = {$IAT/Alarm.Severity2}
      Severity = 2
    [5]:
      Name = Severity3
      Message = {$IAT/Alarm.Severity3}
      Severity = 3
    [6]:
      Name = Severity4
      Message = {$IAT/Alarm.Severity4}
      Severity = 4
    [7]:
      Name = Severity5
      Message = {$IAT/Alarm.Severity5}
      Severity = 5
    [8]:
      Name = Severity1
      Message = {$IAT/Alarm.Severity1}
Element gAlarmXCore_LR_2 (Type=mpalarmxcore)
  mapp.AlarmX.Core:
    BySeverity:
      [0]:
        Severity = 0..100
        [0] = Reaction
          Name = SeverityAnyAlarm
      [1]:
        Severity = 0
        [0] = Reaction
          Name = Severity0
      [2]:
        Severity = 1
        [0] = Reaction
          Name = Severity1
      [3]:
        Severity = 2
        [0] = Reaction
          Name = Severity2
      [4]:
        Severity = 3
        [0] = Reaction
          Name = Severity3
      [5]:
        Severity = 4
        [0] = Reaction
          Name = Severity4
      [6]:
        Severity = 5
        [0] = Reaction
          Name = Severity5
  mapp.AlarmX.Core.Configuration:
    [0]:
      Name = RemMemLost
      Message = {$IAT/Alarm.RemMemLost}
      Code = 1
      Behavior:
        Recording:
          UnacknowledgedToAcknowledged = FALSE
    [1]:
      Name = FileLoadFailed
      Message = {$IAT/Alarm.FileLoadFailed}
      Code = 1001
      Behavior:
        Recording:
          UnacknowledgedToAcknowledged = FALSE
    [2]:
      Name = FileLoadSuccess
      Message = {$IAT/Alarm.FileLoadSuccess}
      Code = 1002
      Behavior:
        Recording:
          UnacknowledgedToAcknowledged = FALSE
    [3]:
      Name = RecipeGeneralError
      Message = {$IAT/Alarm.RecipeGeneralError}
      Code = 1003
      Behavior:
        Recording:
          UnacknowledgedToAcknowledged = FALSE
    [4]:
      Name = Severity2
      Message = {$IAT/Alarm.Severity2}
      Severity = 2
    [5]:
      Name = Severity3
      Message = {$IAT/Alarm.Severity3}
      Severity = 3
    [6]:
      Name = Severity4
      Message = {$IAT/Alarm.Severity4}
      Severity = 4
    [7]:
      Name = Severity5
      Message = {$IAT/Alarm.Severity5}
      Severity = 5
    [8]:
      Name = Severity1
      Message = {$IAT/Alarm.Severity1}
Element gAlarmXCore_LR_1 (Type=mpalarmxcore)
  mapp.AlarmX.Core:
    BySeverity:
      [0]:
        Severity = 0..100
        [0] = Reaction
          Name = SeverityAnyAlarm
      [1]:
        Severity = 0
        [0] = Reaction
          Name = Severity0
      [2]:
        Severity = 1
        [0] = Reaction
          Name = Severity1
      [3]:
        Severity = 2
        [0] = Reaction
          Name = Severity2
      [4]:
        Severity = 3
        [0] = Reaction
          Name = Severity3
      [5]:
        Severity = 4
        [0] = Reaction
          Name = Severity4
      [6]:
        Severity = 5
        [0] = Reaction
          Name = Severity5
  mapp.AlarmX.Core.Configuration:
    [0]:
      Name = RemMemLost
      Message = {$IAT/Alarm.RemMemLost}
      Code = 1
      Behavior:
        Recording:
          UnacknowledgedToAcknowledged = FALSE
    [1]:
      Name = FileLoadFailed
      Message = {$IAT/Alarm.FileLoadFailed}
      Code = 1001
      Behavior:
        Recording:
          UnacknowledgedToAcknowledged = FALSE
    [2]:
      Name = FileLoadSuccess
      Message = {$IAT/Alarm.FileLoadSuccess}
      Code = 1002
      Behavior:
        Recording:
          UnacknowledgedToAcknowledged = FALSE
    [3]:
      Name = RecipeGeneralError
      Message = {$IAT/Alarm.RecipeGeneralError}
      Code = 1003
      Behavior:
        Recording:
          UnacknowledgedToAcknowledged = FALSE
    [4]:
      Name = Severity2
      Message = {$IAT/Alarm.Severity2}
      Severity = 2
    [5]:
      Name = Severity3
      Message = {$IAT/Alarm.Severity3}
      Severity = 3
    [6]:
      Name = Severity4
      Message = {$IAT/Alarm.Severity4}
      Severity = 4
    [7]:
      Name = Severity5
      Message = {$IAT/Alarm.Severity5}
      Severity = 5
    [8]:
      Name = Severity1
      Message = {$IAT/Alarm.Severity1}
Element gAlarmXCore_LR_3 (Type=mpalarmxcore)
  mapp.AlarmX.Core:
    BySeverity:
      [0]:
        Severity = 0..100
        [0] = Reaction
          Name = SeverityAnyAlarm
      [1]:
        Severity = 0
        [0] = Reaction
          Name = Severity0
      [2]:
        Severity = 1
        [0] = Reaction
          Name = Severity1
      [3]:
        Severity = 2
        [0] = Reaction
          Name = Severity2
      [4]:
        Severity = 3
        [0] = Reaction
          Name = Severity3
      [5]:
        Severity = 4
        [0] = Reaction
          Name = Severity4
      [6]:
        Severity = 5
        [0] = Reaction
          Name = Severity5
  mapp.AlarmX.Core.Configuration:
    [0]:
      Name = RemMemLost
      Message = {$IAT/Alarm.RemMemLost}
      Code = 1
      Behavior:
        Recording:
          UnacknowledgedToAcknowledged = FALSE
    [1]:
      Name = FileLoadFailed
      Message = {$IAT/Alarm.FileLoadFailed}
      Code = 1001
      Behavior:
        Recording:
          UnacknowledgedToAcknowledged = FALSE
    [2]:
      Name = FileLoadSuccess
      Message = {$IAT/Alarm.FileLoadSuccess}
      Code = 1002
      Behavior:
        Recording:
          UnacknowledgedToAcknowledged = FALSE
    [3]:
      Name = RecipeGeneralError
      Message = {$IAT/Alarm.RecipeGeneralError}
      Code = 1003
      Behavior:
        Recording:
          UnacknowledgedToAcknowledged = FALSE
    [4]:
      Name = Severity2
      Message = {$IAT/Alarm.Severity2}
      Severity = 2
    [5]:
      Name = Severity3
      Message = {$IAT/Alarm.Severity3}
      Severity = 3
    [6]:
      Name = Severity4
      Message = {$IAT/Alarm.Severity4}
      Severity = 4
    [7]:
      Name = Severity5
      Message = {$IAT/Alarm.Severity5}
      Severity = 5
    [8]:
      Name = Severity1
      Message = {$IAT/Alarm.Severity1}
Element gAlarmXCore_Global (Type=mpalarmxcore)
  mapp.AlarmX.Core:
    BySeverity:
      [0]:
        Severity = 0..100
        [0] = Reaction
          Name = SeverityAnyAlarm
      [1]:
        Severity = 0
        [0] = Reaction
          Name = Severity0
      [2]:
        Severity = 1
        [0] = Reaction
          Name = Severity1
      [3]:
        Severity = 2
        [0] = Reaction
          Name = Severity2
      [4]:
        Severity = 3
        [0] = Reaction
          Name = Severity3
      [5]:
        Severity = 4
        [0] = Reaction
          Name = Severity4
      [6]:
        Severity = 5
        [0] = Reaction
          Name = Severity5
  mapp.AlarmX.Core.Configuration:
    [0]:
      Name = RemMemLost
      Message = {$IAT/Alarm.RemMemLost}
      Code = 1
      Behavior:
        Recording:
          UnacknowledgedToAcknowledged = FALSE
    [1]:
      Name = FileLoadFailed
      Message = {$IAT/Alarm.FileLoadFailed}
      Code = 1001
      Behavior:
        Recording:
          UnacknowledgedToAcknowledged = FALSE
    [2]:
      Name = FileLoadSuccess
      Message = {$IAT/Alarm.FileLoadSuccess}
      Code = 1002
      Behavior:
        Recording:
          UnacknowledgedToAcknowledged = FALSE
    [3]:
      Name = RecipeGeneralError
      Message = {$IAT/Alarm.RecipeGeneralError}
      Code = 1003
      Behavior:
        Recording:
          UnacknowledgedToAcknowledged = FALSE
    [4]:
      Name = Severity2
      Message = {$IAT/GlobalAlarm.Severity2}
      Severity = 2
    [5]:
      Name = Severity3
      Message = {$IAT/GlobalAlarm.Severity3}
      Severity = 3
    [6]:
      Name = Severity4
      Message = {$IAT/GlobalAlarm.Severity4}
      Severity = 4
    [7]:
      Name = Severity5
      Message = {$IAT/GlobalAlarm.Severity5}
      Severity = 5
    [8]:
      Name = Severity1
      Message = {$IAT/GlobalAlarm.Severity1}
Element gAlarmXCore_LR_0 (Type=mpalarmxcore)
  mapp.AlarmX.Core:
    BySeverity:
      [0]:
        Severity = 0..100
        [0] = Reaction
          Name = SeverityAnyAlarm
      [1]:
        Severity = 0
        [0] = Reaction
          Name = Severity0
      [2]:
        Severity = 1
        [0] = Reaction
          Name = Severity1
      [3]:
        Severity = 2
        [0] = Reaction
          Name = Severity2
      [4]:
        Severity = 3
        [0] = Reaction
          Name = Severity3
      [5]:
        Severity = 4
        [0] = Reaction
          Name = Severity4
      [6]:
        Severity = 5
        [0] = Reaction
          Name = Severity5
  mapp.AlarmX.Core.Configuration:
    [0]:
      Name = RemMemLost
      Message = {$IAT/Alarm.RemMemLost}
      Code = 1
      Behavior:
        Recording:
          UnacknowledgedToAcknowledged = FALSE
    [1]:
      Name = FileLoadFailed
      Message = {$IAT/Alarm.FileLoadFailed}
      Code = 1001
      Behavior:
        Recording:
          UnacknowledgedToAcknowledged = FALSE
    [2]:
      Name = FileLoadSuccess
      Message = {$IAT/Alarm.FileLoadSuccess}
      Code = 1002
      Behavior:
        Recording:
          UnacknowledgedToAcknowledged = FALSE
    [3]:
      Name = RecipeGeneralError
      Message = {$IAT/Alarm.RecipeGeneralError}
      Code = 1003
      Behavior:
        Recording:
          UnacknowledgedToAcknowledged = FALSE
    [4]:
      Name = Severity2
      Message = {$IAT/Alarm.Severity2}
      Severity = 2
    [5]:
      Name = Severity3
      Message = {$IAT/Alarm.Severity3}
      Severity = 3
    [6]:
      Name = Severity4
      Message = {$IAT/Alarm.Severity4}
      Severity = 4
    [7]:
      Name = Severity5
      Message = {$IAT/Alarm.Severity5}
      Severity = 5
    [8]:
      Name = Severity1
      Message = {$IAT/Alarm.Severity1}
```

### Config_2.mpalarmxhistory - 5APC3100_KBU3_000/mappServices/Config_2.mpalarmxhistory
```
Element gAlarmXHistory (Type=mpalarmxhistory)
  mapp.AlarmX.History:
    Export:
      FileNamePattern = AlarmHistory/Alarms_%Y_%m_%d_%H_%M_%S.csv
    Memory:
      MemorySize = 5
      BufferSize = 1
```

### Config_3.mpcomgroup - 5APC3100_KBU3_000/mappServices/Config_3.mpcomgroup
```
Element gGroup_LR_0 (Type=mpcomgroup)
  Linking:
    Subnodes:
      0 = gAlarmXCore_LR_0
      1 = gAlarmXHistory_LR_0
  Alarms = MpAlarmX
Element gGroup_LR_1 (Type=mpcomgroup)
  Linking:
    Subnodes:
      0 = gAlarmXCore_LR_1
      1 = gAlarmXHistory_LR_1
  Alarms = MpAlarmX
Element gGroup_LR_10 (Type=mpcomgroup)
  Linking:
    Subnodes:
      0 = gAlarmXCore_LR_10
      1 = gAlarmXHistory_LR_10
  Alarms = MpAlarmX
Element gGroup_LR_11 (Type=mpcomgroup)
  Linking:
    Subnodes:
      0 = gAlarmXCore_LR_11
      1 = gAlarmXHistory_LR_11
  Alarms = MpAlarmX
Element gGroup_LR_12 (Type=mpcomgroup)
  Linking:
    Subnodes:
      0 = gAlarmXCore_LR_12
      1 = gAlarmXHistory_LR_12
  Alarms = MpAlarmX
Element gGroup_LR_20 (Type=mpcomgroup)
  Linking:
    Subnodes:
      0 = gAlarmXCore_LR_20
      1 = gAlarmXHistory_LR_20
  Alarms = MpAlarmX
Element gGroup_LR_21 (Type=mpcomgroup)
  Linking:
    Subnodes:
      0 = gAlarmXCore_LR_21
      1 = gAlarmXHistory_LR_21
  Alarms = MpAlarmX
Element gGroup_LR_22 (Type=mpcomgroup)
  Linking:
    Subnodes:
      0 = gAlarmXCore_LR_22
      1 = gAlarmXHistory_LR_22
  Alarms = MpAlarmX
Element gGroup_LR_23 (Type=mpcomgroup)
  Linking:
    Subnodes:
      0 = gAlarmXCore_LR_23
      1 = gAlarmXHistory_LR_23
  Alarms = MpAlarmX
Element gGroup_LR_24 (Type=mpcomgroup)
  Linking:
    Subnodes:
      0 = gAlarmXCore_LR_24
      1 = gAlarmXHistory_LR_24
  Alarms = MpAlarmX
Element gGroup_LR_25 (Type=mpcomgroup)
  Linking:
    Subnodes:
      0 = gAlarmXCore_LR_25
      1 = gAlarmXHistory_LR_25
  Alarms = MpAlarmX
Element gGroup_LR_19 (Type=mpcomgroup)
  Linking:
    Subnodes:
      0 = gAlarmXCore_LR_19
      1 = gAlarmXHistory_LR_19
  Alarms = MpAlarmX
Element gGroup_LR_18 (Type=mpcomgroup)
  Linking:
    Subnodes:
      0 = gAlarmXCore_LR_18
      1 = gAlarmXHistory_LR_18
  Alarms = MpAlarmX
Element gGroup_LR_17 (Type=mpcomgroup)
  Linking:
    Subnodes:
      0 = gAlarmXCore_LR_17
      1 = gAlarmXHistory_LR_17
  Alarms = MpAlarmX
Element gGroup_LR_16 (Type=mpcomgroup)
  Linking:
    Subnodes:
      0 = gAlarmXCore_LR_16
      1 = gAlarmXHistory_LR_16
  Alarms = MpAlarmX
Element gGroup_LR_15 (Type=mpcomgroup)
  Linking:
    Subnodes:
      0 = gAlarmXCore_LR_15
      1 = gAlarmXHistory_LR_15
  Alarms = MpAlarmX
Element gGroup_LR_14 (Type=mpcomgroup)
  Linking:
    Subnodes:
      0 = gAlarmXCore_LR_14
      1 = gAlarmXHistory_LR_14
  Alarms = MpAlarmX
Element gGroup_LR_13 (Type=mpcomgroup)
  Linking:
    Subnodes:
      0 = gAlarmXCore_LR_13
      1 = gAlarmXHistory_LR_13
  Alarms = MpAlarmX
Element gGroup_LR_2 (Type=mpcomgroup)
  Linking:
    Subnodes:
      0 = gAlarmXCore_LR_2
      1 = gAlarmXHistory_LR_2
  Alarms = MpAlarmX
Element gGroup_LR_3 (Type=mpcomgroup)
  Linking:
    Subnodes:
      0 = gAlarmXCore_LR_3
      1 = gAlarmXHistory_LR_3
  Alarms = MpAlarmX
Element gGroup_LR_4 (Type=mpcomgroup)
  Linking:
    Subnodes:
      0 = gAlarmXCore_LR_4
      1 = gAlarmXHistory_LR_4
  Alarms = MpAlarmX
Element gGroup_LR_5 (Type=mpcomgroup)
  Linking:
    Subnodes:
      0 = gAlarmXCore_LR_5
      1 = gAlarmXHistory_LR_5
  Alarms = MpAlarmX
Element gGroup_LR_6 (Type=mpcomgroup)
  Linking:
    Subnodes:
      0 = gAlarmXCore_LR_6
      1 = gAlarmXHistory_LR_6
  Alarms = MpAlarmX
Element gGroup_LR_7 (Type=mpcomgroup)
  Linking:
    Subnodes:
      0 = gAlarmXCore_LR_7
      1 = gAlarmXHistory_LR_7
  Alarms = MpAlarmX
Element gGroup_LR_8 (Type=mpcomgroup)
  Linking:
    Subnodes:
      0 = gAlarmXCore_LR_8
      1 = gAlarmXCore_LR_8
  Alarms = MpAlarmX
Element gGroup_LR_9 (Type=mpcomgroup)
  Linking:
    Subnodes:
      0 = gAlarmXCore_LR_9
      1 = gAlarmXCore_LR_9
  Alarms = MpAlarmX
Element gGroup_Global (Type=mpcomgroup)
  Linking:
    Subnodes:
      0 = gAlarmXCore_Global
  Alarms = MpAlarmX
```

## Configuration Config1

CPU PC_any, AutomationRuntime J4.93, Build 4.1.2, Safety 0.0, Vc V4.73.2

### Task classes (Cpu.sw)
```
Cyclic#1 (cycle 10000 us, tolerance 0 us):
  Main <- Main.prg
  ModbusDriv <- ModbusDriver.prg
Libraries: AsOpcUas, AsOpcUac, runtime, Acp10man, Acp10par, NcGlobal, standard
```

### Hardware
```
PC : PC_any v1.1.1.0 (OrderNumber=PC)
  Connector IF3:
    InternetAddress = 172.16.1.63
    ActivateModbus = 1
    NumSlaves = -1
    NumAllBlocks = -1
    MemSizeIn = -1
    MemSizeOut = -1
    SlaveDiagnostics = 1
  ConfigurationID = RemoteVis_CleanChemistry_Config1
  VolatileGlobalPvSize = 655350
  Cyclic1Duration = 10000
  Cyclic1Tolerance = 0
  FileDevice1
  FileDeviceName1 = USER
  FileDevicePath1 = USER_PATH
  ActivateOpcUa = 1
  OpcUaInformationModels_PV_Version = 1
```

### Acp10cfg.ncc - PC/Acp10cfg.ncc
```
NcConfiguration (Version=3.13.1, NcSwId=Acp10)
  ACP10CF1_typ:
    cnt_nettrc_rec_drive = 150
    bufsize_trace_upload = 1200
    tc_nc_man_task = Cyclic #1
    glob_pv_as_ncobject = Yes
    ncsys_dl_broadcast = Yes
    ncsys_dl_acp_reset = Yes
    safemc_log_err_to_ax = Yes
    network_init:
      ncsw_init_execute = Yes
      automatic_execute = No
      node_nr_warning = Yes
      net_err_before_ncact = Yes
    nettrc:
      enter_parsecrec = Yes
      enter_ncaction = Yes
      save_ring_startidx = No
    cam_prof_download:
      cam_dat_dl_parallel = No
      tc_cam_dl_parallel = Task class for NC Manager task
```

### Config_1.mpalarmxcore - PC/mappServices/Config_1.mpalarmxcore
```
Element gAlarmXCore (Type=mpalarmxcore)
  mapp.AlarmX.Core:
    BySeverity:
      [0]:
        Severity = 0..100
        [0] = Reaction
          Name = SeverityAnyAlarm
      [1]:
        Severity = 0
        [0] = Reaction
          Name = Severity0
      [2]:
        Severity = 1
        [0] = Reaction
          Name = Severity1
      [3]:
        Severity = 2
        [0] = Reaction
          Name = Severity2
      [4]:
        Severity = 3
        [0] = Reaction
          Name = Severity3
      [5]:
        Severity = 4
        [0] = Reaction
          Name = Severity4
      [6]:
        Severity = 5
        [0] = Reaction
          Name = Severity5
  mapp.AlarmX.Core.Configuration:
    [0]:
      Name = RemMemLost
      Message = {$IAT/Alarm.RemMemLost}
      Code = 1000
      Behavior:
        Recording:
          UnacknowledgedToAcknowledged = FALSE
    [1]:
      Name = FileLoadFailed
      Message = {$IAT/Alarm.FileLoadFailed}
      Code = 1001
      Behavior:
        Recording:
          UnacknowledgedToAcknowledged = FALSE
    [2]:
      Name = FileLoadSuccess
      Message = {$IAT/Alarm.FileLoadSuccess}
      Code = 1002
      Behavior:
        Recording:
          UnacknowledgedToAcknowledged = FALSE
    [3]:
      Name = RecipeGeneralError
      Message = {$IAT/Alarm.RecipeGeneralError}
      Code = 1003
      Behavior:
        Recording:
          UnacknowledgedToAcknowledged = FALSE
    [4]:
      Name = MonitorConvInOverflow
      Message = {$IAT/Alarm.MonitorConvInOverflow}
      Code = 9001
      Severity = 2
      Behavior:
        Recording:
          UnacknowledgedToAcknowledged = FALSE
    [5]:
      Name = MonitorConvInOverflowNoHigh
      Message = {$IAT/Alarm.MonitorConvInOverflowNoHigh}
      Code = 9002
      Severity = 2
      Behavior:
        Recording:
          UnacknowledgedToAcknowledged = FALSE
    [6]:
      Name = MonitorConvInLowNoPresent
      Message = {$IAT/Alarm.MonitorConvInLowNoPresent}
      Code = 9003
      Severity = 2
      Behavior:
        Recording:
          UnacknowledgedToAcknowledged = FALSE
    [7]:
      Name = MonitorConvInHighNoLow
      Message = {$IAT/Alarm.MonitorConvInHighNoLow}
      Code = 9004
      Severity = 2
      Behavior:
        Recording:
          UnacknowledgedToAcknowledged = FALSE
    [8]:
      Name = MonitorConvInNoFeedback
      Message = {$IAT/Alarm.MonitorConvInNoFeedback}
      Code = 9005
      Severity = 2
      Behavior:
        Recording:
          UnacknowledgedToAcknowledged = FALSE
    [9]:
      Name = MonitorWheelNoFeedback
      Message = {$IAT/Alarm.MonitorWheelNoFeedback}
      Code = 9006
      Severity = 2
      Behavior:
        Recording:
          UnacknowledgedToAcknowledged = FALSE
    [10]:
      Name = MonitorE_STOP
      Message = {$IAT/Alarm.MonitorHMI_STOP}
      Code = 9998
      Severity = 5
      Behavior:
        Recording:
          UnacknowledgedToAcknowledged = FALSE
    [11]:
      Name = MonitorHMI_STOP
      Message = {$IAT/Alarm.MonitorHMI_STOP}
      Code = 9999
      Severity = 4
      Behavior:
        Recording:
          UnacknowledgedToAcknowledged = FALSE
    [12]:
      Name = MasterExternalPause
      Message = {$IAT/Alarm.MasterExternalPause}
      Code = 1113
      Behavior:
        Recording:
          UnacknowledgedToAcknowledged = FALSE
    [13]:
      Name = MasterExternalControlledStop
      Message = {$IAT/Alarm.MasterExternalControlledStop}
      Code = 1114
      Severity = 3
      Behavior:
        Recording:
          UnacknowledgedToAcknowledged = FALSE
    [14]:
      Name = MasterExternalUncontrolledStop
      Message = {$IAT/Alarm.MasterExternalUncontrolledStop}
      Code = 1115
      Severity = 4
      Behavior:
        Recording:
          UnacknowledgedToAcknowledged = FALSE
```

## Configuration Config2

CPU X20CP1584, AutomationRuntime J4.93, Build 4.1.2, Safety 0.0, Vc V4.73.2

### Hardware
```
X20CP1584 : X20CP1584 v1.10.0.0
  Connector IF1:
    ActivateIna = 0
  Connector IF2:
    ActivateDevice = 1
    Mode = Manual
    InternetAddress = 172.16.1.63
    SubnetMask = 255.255.255.0
    InaPort = 11160
    ActivateSnmp = 2
    ActivateModbus = 1
    NumSlaves = -1
    NumAllBlocks = -1
    MemSizeIn = -1
    MemSizeOut = -1
    SlaveDiagnostics = 1
  ConfigurationID = RemoteVis_CleanChemistry_Config1
  VolatileGlobalPvSize = 655350
  Cyclic1Tolerance = 0
  FileDevice1
  FileDeviceName1 = USER
  FileDevicePath1 = USER_PATH
  ActivateOpcUa = 1
  OpcUaInformationModels_PV_Version = 1
```

## Configuration PC

CPU PC_any, AutomationRuntime J4.93, Build 4.1.2, Safety 0.0, Vc V4.73.2

### Task classes (Cpu.sw)
```
Cyclic#1:
  Master_LR <- modbusTCP.Master_LR.prg
  ModbusDriv <- (binary)
Cyclic#2:
  Vis <- Vis.prg
DataObjects: Acp10sys
Binaries: FWRules, TCData, mvLoader, udbdef, TCLang, acp10cfg, arnc0cfg, Acp10map, iomap, arconfig, asfw, ashwac, sysconf, User, Role, ashwd, TC
Libraries: AsOpcUas, AsOpcUac, runtime, NcGlobal, standard, MbusTCP, IDEC_Real, astime, AsIecCon, AsTCP, AsBrStr, AsARCfg, sys_lib, ArTextSys, Str2DtPvdr, powerlnk, arssl, asstring, AsBrWStr, MpCom, MpBase, HA, HA_Version, HA_IO, HA_Dir, HA_Convert, HA_AlarmX, HA_ItemX, HA_RAND, ArEventLog, ArProject, brsystem, FileIO, AsUSB, HA_Array, HA_SysErr
```

## Logical view

Binary libraries used (declarations not repeated): operator, runtime, astime, AsIecCon, AsOpcUas, AsOpcUac, NcGlobal 3.13.1, standard, AsTCP, AsBrStr, AsARCfg, sys_lib, ArTextSys, asstring, AsBrWStr, MpBase, ArEventLog, ArProject, brsystem, FileIO, AsUSB, AsHttp, AsICMP, AsHost, ArUser, MpUserX 5.24.5, MpCom 5.24.5, AsIODiag, MpAlarmX 5.24.5, MpRecipe 5.24.5, MpServer

### Global.var - Global variables
```iecst
VAR
	RecipeLoaded : BOOL := FALSE;
	RECIPE_LR_TEMP : {REDUND_UNREPLICABLE} ARRAY[0..MAX_SKIDS_LR] OF Recipe_type := [18((0))];
	CONTACT_NAMES : {REDUND_UNREPLICABLE} ARRAY[0..MAX_SKIDS_LR] OF STRING[80];
	gRecipe_LR : {REDUND_UNREPLICABLE} ARRAY[0..MAX_SKIDS_LR] OF Recipe_type := [(Notes:='Test PLC'),(Notes:='GA101 - Claxton - Sylvania'),2(0),(Notes:='AL100 - Teleios - Ala Trade Boaz'),(Notes:='OK110 - Teleios - Tyson Broken Bow'),(Notes:='AR100 - Teleios - Twin Rivers Foods Ft. Smith'),(Notes:='TX575 - Teleios - Pilgrim Pride Nacogdoches'),(Notes:='OK110 - Teleios - Tyson Broken Bow'),0,(Notes:='TX575 - Teleios - Pilgrim Pride Nacogdoches'),(Notes:='GA101 - Claxton - Sylvania'),(Notes:='LA113 - Teleios - Wayne Sanderson Farms Hammond'),0,(Notes:='OK110 - Teleios - Tyson Broken Bow'),(Notes:='AR101 - Teleios - Custom Craft Batesville'),2(0)];
	gServices : Services_typ := (0);
	SkidID : USINT := 0;
	gModbus_LR : ARRAY[0..MAX_SKIDS_LR] OF Modbus_Type := [(0)];
	gCMD_HR : ARRAY[0..MAX_SKIDS_HR] OF CMD_Type := [(0)];
	gCMD_LR : ARRAY[0..MAX_SKIDS_LR] OF CMD_Type := [(0)];
	gModbus_HR : ARRAY[0..MAX_SKIDS_HR] OF Modbus_Type := [(0)];
	gSkid_LR : ARRAY[0..MAX_SKIDS_LR] OF Skid_type := [(0)];
	gSkid_HR : ARRAY[0..MAX_SKIDS_HR] OF Skid_type := [(0)];
	gVis : Vis_Type := (0);
	gUnit_HR : ARRAY[0..MAX_SKIDS_HR] OF UINT := [(0)];
	gUnit_LR : ARRAY[0..MAX_SKIDS_LR] OF UINT := [(0)];
	gAlarmAddData_Global : HA_AlarmX_AlarmExtraData_typ := (0);
	gAlarmAddData : HA_AlarmX_AlarmExtraData_typ := (0);
	gErrorReset : BOOL := FALSE;
END_VAR
```

### Constants.var
```iecst
VAR CONSTANT
	MAX_CLIENTS : USINT := 10;
	P102_LS_TRIGGER : USINT := 70; (*% To Trigger P102 LS*)
	P103_LS_TRIGGER : USINT := 70; (*% To Trigger P103 LS*)
	LSHH200_TRIGGER : USINT := 70; (*% To Trigger BT HH Indicator*)
	BT_VOLUME : UDINT := 1060; (*Buffer Tank Volume, ml*)
	MAX_SKIDS_HR : USINT := 0;
	MAX_SKIDS_LR : USINT := 22;
	MAX_MODBUS_BLOCKS : USINT := 140;
	SLAVE_IP_ADDRESSES_HR : ARRAY[0..MAX_SKIDS_HR] OF STRING[20] := ['172.16.1.122'];
	SLAVE_IP_ADDRESSES_LR : ARRAY[0..MAX_SKIDS_LR] OF STRING[20] := ['172.16.1.101','172.16.1.103','172.16.1.104','172.16.1.112','172.16.1.105','172.16.1.108','172.16.1.110','172.16.1.111','172.16.1.106','172.16.1.114','172.16.1.118','172.16.1.113','172.16.1.117','172.16.1.128','172.16.1.116','172.16.1.127','172.16.1.121','172.16.1.129','172.16.1.124','172.16.1.119','172.16.1.126','172.16.1.132','172.16.1.123'];
	MAX_CONTACTS : USINT := 7;
END_VAR
```
